// TIA Portal V20 export
// export: Created 2025-12-01T14:56:22.1165427Z, ExportSetting None, DisplayName Totally Integrated Automation Portal, DisplayVersion V20 Update 3, DisplayName TIA Portal Openness, DisplayVersion V20 Update 3, DisplayName TIA Portal Version Control Interface, DisplayVersion V20 Update 3, DisplayName STEP 7 Professional, DisplayVersion V20 Update 3, DisplayName STEP 7 Safety, DisplayVersion V20 Update 2, DisplayName WinCC Basic/Comfort/Advanced, DisplayVersion V20 Update 3, DisplayName WinCC Professional, DisplayVersion V20 Update 3, DisplayName WinCC Unified, DisplayVersion V20 Update 3
TYPE "NDD_Interlock_TElev"
   STRUCT
      PeticionEntrada : Bool;
      PermisoEntradaPaleta : Bool;
      PermisoSalidaPaleta : Bool;
      OrdenTELEV_S0 : Bool;
      FinOrdenTELEV_S0 : Bool;
      OrdenTELEV_S3 : Bool;
      OrdenTELEV_S1 : Bool;
      FinOrdenTELEV_S13 : Bool;
      AVTF_Entrada : Bool;
      PTF_Entrada : Bool;
      FTF_Entrada : Bool;
      AVTF_Salida : Bool;
      PTF_Salida : Bool;
      FTF_Salida : Bool;
      DesCargaAct_Entrada : Bool;
      DesCargaAct_Salida : Bool;
      ConCarga_TELEV : Bool;
      Libre_21 : Bool;
      Libre_22 : Bool;
      Libre_23 : Bool;
      Libre_24 : Bool;
      Libre_25 : Bool;
      Libre_26 : Bool;
      Libre_27 : Bool;
      TELEV_EnReset { ExternalVisible := 'False'} : Bool;
      TELEV_EnCarga { ExternalVisible := 'False'} : Bool;
      TELEV_EnVacio : Bool;
      TELEV_Entrando_E1 : Bool;
      TELEV_Saliendo_S3 : Bool;
      TELEV_Entrando_E2 : Bool;
      TELEV_Saliendo_S2 : Bool;
      Libre_37 : Bool;
   END_STRUCT;
END_TYPE
